{attribute 'qualified_only'}
VAR_GLOBAL
 DA: ARRAY[0..1023] OF BYTE;
END_VAR

(* stored: Version 1.1.0.1, ProductVersion 3.1.4024.5
   GVL DigOutput: Id {860fb756-d094-44f6-895d-8e627f205f5e} *)
